# EPICS autosave request: CARSApp/Db/mirror_pid_control_settings.req
# FILE... mirror_pid_control_settings.req
file "pid_control_settings.req", P=$(P), PID=$(PID)
file "transform_settings.req", P=$(P)$(PID)_incalc
